INTERFACE PUBLIC I_SuspendedCommands

METHOD PUBLIC Abort
END_METHOD

METHOD PUBLIC Stop
END_METHOD

METHOD PUBLIC Unsuspend
END_METHOD

END_INTERFACE

(* stored: Version 1.1.0.1, ProductVersion 3.1.4026.6
   Itf I_SuspendedCommands: Id {f31c0d5b-acac-0491-1bc4-9e5110404f07}
   Method Abort: Id {9134edc0-35df-4e22-9894-227f597c7f41}
   Method Stop: Id {f55dc1d3-4853-4e42-ad1b-4354fd287f20}
   Method Unsuspend: Id {199c3e50-b73d-0b1c-0fc2-c7e590019e1b} *)
